// TIA Portal project "project A" (V18)
// Youtube part 1

(* hardware
DEVICE "S7-1500/ET200MP station_1"  S7-1500 station
   slot 0: "Rail_0"  Rack  6ES7 590-1***0-0AA0
   slot 1: "Brain"  CPU 1512C-1 PN  6ES7 512-1CK00-0AB0  V1.8
      slot 3: "CPU display_1"  6ES7591-1AA00-0AA0
      slot 32768: "PROFINET interface_1"  X1
         slot 32769: "Port_1"  X1 P1
         slot 32770: "Port_2"  X1 P2
   slot 2: "DI 16x24VDC / DQ 16x24VDC/0.5A BA_1"  DI 16x24VDC/DQ 16x24VDC/0.5A BA  6ES7 523-1BL00-0AA0  V1.1
*)

// ===== PLC "Brain"  CPU 1512C-1 PN =====

VAR_GLOBAL   // PLC tag table "Conveyor1"
   "B1" AT %I10.0 : Bool;   // Component at conveyor start
   "B2" AT %I10.1 : Bool;   // Component at conveyor center
   "B3" AT %I10.2 : Bool;   // No component at conveyor end
   "S1" AT %I10.3 : Bool;   // Start button
   "K1" AT %Q4.0 : Bool;   // Conveyor belt on
   "1M1" AT %Q4.1 : Bool;   // Open stopper
   "P1" AT %Q4.2 : Bool;   // Indicator LED
END_VAR

VAR_GLOBAL   // PLC tag table "Clock Memory"
   "Clock_Byte" AT %MB0 : Byte;
   "Clock_10Hz" AT %M0.0 : Bool;
   "Clock_5Hz" AT %M0.1 : Bool;
   "Clock_2.5Hz" AT %M0.2 : Bool;
   "Clock_2Hz" AT %M0.3 : Bool;
   "Clock_1.25Hz" AT %M0.4 : Bool;
   "Clock_1Hz" AT %M0.5 : Bool;
   "Clock_0.625Hz" AT %M0.6 : Bool;
   "Clock_0.5Hz" AT %M0.7 : Bool;
END_VAR

VAR_GLOBAL   // PLC tag table "Conveyor2"
   "B4" AT %I11.0 : Bool;   // Component at conveyor start
   "B5" AT %I11.1 : Bool;   // Component at conveyor center
   "B6" AT %I11.2 : Bool;   // No component at conveyor end
   "K2" AT %Q5.0 : Bool;   // Conveyor belt on
   "2M1" AT %Q5.1 : Bool;   // Open stopper
   "P2" AT %Q5.2 : Bool;   // Indicator LED
END_VAR

FUNCTION "Conveyor" : Void   // FC1, LAD
{ S7_Optimized_Access := 'TRUE' }
VERSION : 0.1
   VAR_INPUT
      "Conveyor Start" : Bool;
      "Conveyor Center" : Bool;
      "Conveyor End" : Bool;
      "Start Button" : Bool;
      "Conveyor On Frequency" : Bool;
      "Part at Start Frequency" : Bool;
   END_VAR
   VAR_OUTPUT
      Stopper : Bool;
      LED : Bool;
   END_VAR
   VAR_IN_OUT
      Conveyor : Bool;
   END_VAR
BEGIN

REGION Network 1: conveyor bellt
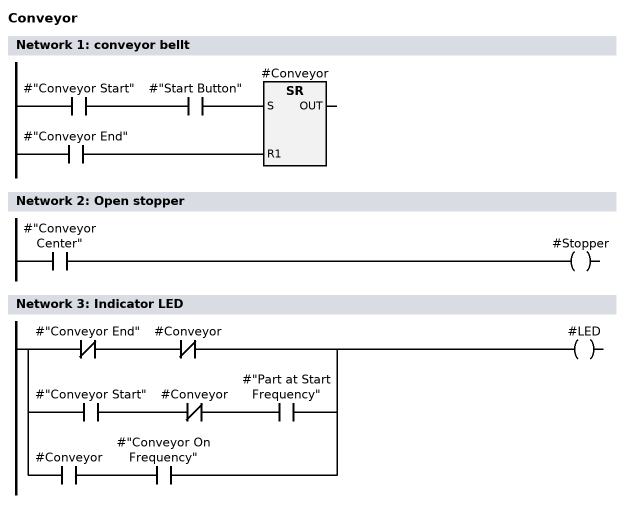
   RUNG wire#powerrail
      Contact( #"Conveyor Start" )
      Contact( #"Start Button" )
      S_SR(operand := #Conveyor, r1 := wire#w1)
   END_RUNG
   RUNG wire#powerrail
      Contact( #"Conveyor End" )
   END_RUNG wire#w1
   // the same network as SCL:
   IF #"Conveyor Start" AND #"Start Button" THEN
       #Conveyor := TRUE;   // SR flip-flop
   END_IF;
   IF #"Conveyor End" THEN #Conveyor := FALSE; END_IF;
END_REGION

REGION Network 2: Open stopper
   RUNG wire#powerrail
      Contact( #"Conveyor Center" )
      Coil( #Stopper )
   END_RUNG
   // the same network as SCL:
   #Stopper := #"Conveyor Center";
END_REGION

REGION Network 3: Indicator LED
   RUNG wire#powerrail
      I_Contact( #"Conveyor End" )
      I_Contact( #Conveyor )
      wire#w1
      Coil( #LED )
   END_RUNG
   RUNG wire#powerrail
      Contact( #"Conveyor Start" )
      I_Contact( #Conveyor )
      Contact( #"Part at Start Frequency" )
   END_RUNG wire#w1
   RUNG wire#powerrail
      Contact( #Conveyor )
      Contact( #"Conveyor On Frequency" )
   END_RUNG wire#w1
   // the same network as SCL:
   #LED := (NOT #"Conveyor End" AND NOT #Conveyor) OR (#"Conveyor Start" AND NOT #Conveyor AND #"Part at Start Frequency") OR (#Conveyor AND #"Conveyor On Frequency");
END_REGION
END_FUNCTION

ORGANIZATION_BLOCK "Main"   // OB1, LAD, ProgramCycle
TITLE = "Main Program Sweep (Cycle)"
{ S7_Optimized_Access := 'TRUE' }
VERSION : 0.1
   VAR_INPUT
      Initial_Call : Bool;   // Initial call of this OB
      Remanence : Bool;   // =True, if remanent data are available
   END_VAR
BEGIN

REGION Network 1: Function call Conveyor
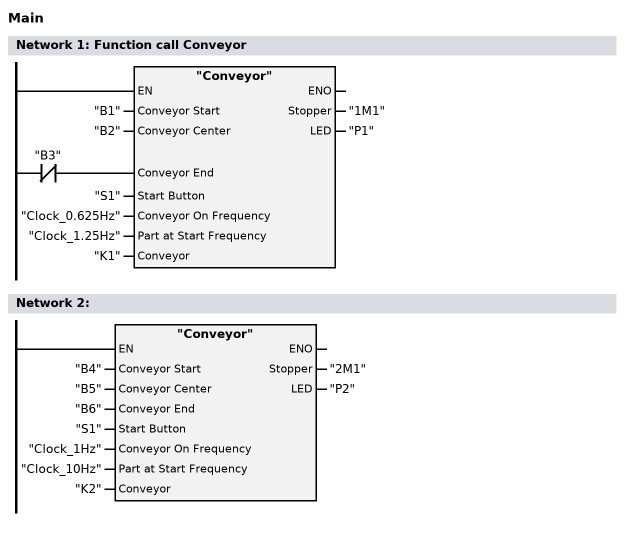
   RUNG wire#powerrail
      "Conveyor"("Conveyor End" := wire#w1, "Conveyor Start" := "B1", "Conveyor Center" := "B2", "Start Button" := "S1", "Conveyor On Frequency" := "Clock_0.625Hz", "Part at Start Frequency" := "Clock_1.25Hz", Conveyor := "K1", Stopper => "1M1", LED => "P1")
   END_RUNG
   RUNG wire#powerrail
      I_Contact( "B3" )
   END_RUNG wire#w1
   // the same network as SCL:
   "Conveyor"("Conveyor Start" := "B1",
              "Conveyor Center" := "B2",
              "Conveyor End" := NOT "B3",
              "Start Button" := "S1",
              "Conveyor On Frequency" := "Clock_0.625Hz",
              "Part at Start Frequency" := "Clock_1.25Hz",
              Conveyor := "K1",
              Stopper => "1M1",
              LED => "P1");
END_REGION

REGION Network 2
   RUNG wire#powerrail
      "Conveyor"("Conveyor Start" := "B4", "Conveyor Center" := "B5", "Conveyor End" := "B6", "Start Button" := "S1", "Conveyor On Frequency" := "Clock_1Hz", "Part at Start Frequency" := "Clock_10Hz", Conveyor := "K2", Stopper => "2M1", LED => "P2")
   END_RUNG
   // the same network as SCL:
   "Conveyor"("Conveyor Start" := "B4",
              "Conveyor Center" := "B5",
              "Conveyor End" := "B6",
              "Start Button" := "S1",
              "Conveyor On Frequency" := "Clock_1Hz",
              "Part at Start Frequency" := "Clock_10Hz",
              Conveyor := "K2",
              Stopper => "2M1",
              LED => "P2");
END_REGION
END_ORGANIZATION_BLOCK